Staubli VAL3: start.pgx

program start()
begin

  // Library to handle all of the interface actions for CS9 controller
  // Loaded at runtime in ros_server()

  // DO NOT auto-load
  // Auto-loading will break cross-controller functionality
  // The correct library will be loaded at runtime, otherwise an error will be generated

end
